// TIA Portal V15.1 export
// export: Created 2024-06-21T08:41:25.4338314Z, ExportSetting WithDefaults, DisplayName Totally Integrated Automation Portal, DisplayVersion V15.1 Update 5, DisplayName TIA Portal Openness, DisplayVersion V15.1 Update 5, DisplayName SINAMICS Startdrive Advanced, DisplayVersion V15.1, DisplayName G130, G150, S120, S150, SINAMICS MV, S210, DisplayVersion V15.1, DisplayName G110M, G120, G120C, G120D, G120P, DisplayVersion V15.1, DisplayName STEP 7 Professional, DisplayVersion V15.1 Update 5, DisplayName STEP 7 Safety, DisplayVersion V15.1, DisplayName WinCC Professional, DisplayVersion V15.1 Update 5, DisplayName SIMATIC Visualization Architect, DisplayVersion V15.1
FUNCTION "209000NCP01ComSafety" : Void   // FC199, FBD
TITLE = 209000NCP01ComSafety
{ S7_Optimized_Access := 'TRUE' }
VERSION : 0.1
// stored: AutoNumber false, IsIECCheckEnabled false, SetENOAutomatically False, UDAEnableTagReadback false
BEGIN

REGION Network 1: **** 5.2 - Equations **** 209230ASD01 Alarm Reset PB
   // Alarm Reset Push Button of MGB
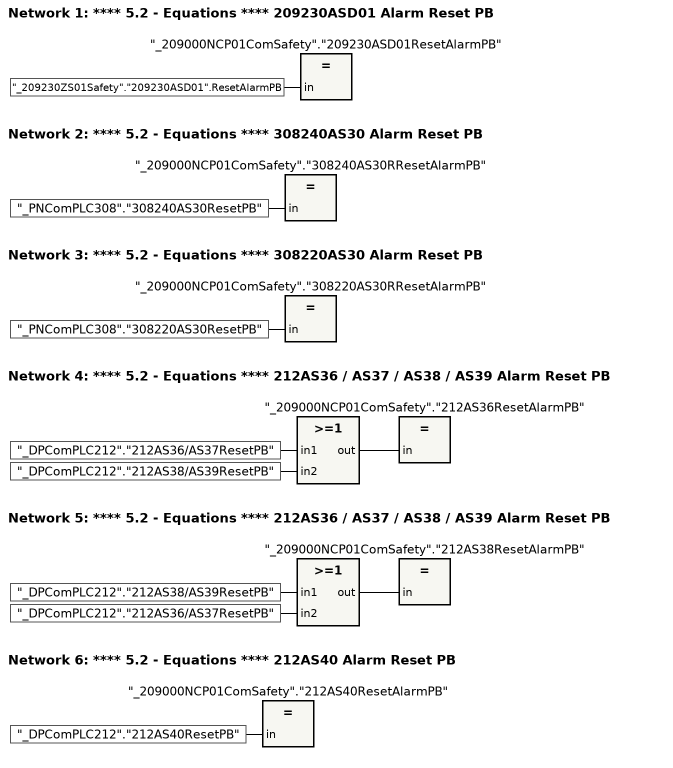
   "_209000NCP01ComSafety"."209230ASD01ResetAlarmPB" := "_209230ZS01Safety"."209230ASD01".ResetAlarmPB;
END_REGION

REGION Network 2: **** 5.2 - Equations **** 308240AS30 Alarm Reset PB
   "_209000NCP01ComSafety"."308240AS30RResetAlarmPB" := "_PNComPLC308"."308240AS30ResetPB";
END_REGION

REGION Network 3: **** 5.2 - Equations **** 308220AS30 Alarm Reset PB
   "_209000NCP01ComSafety"."308220AS30RResetAlarmPB" := "_PNComPLC308"."308220AS30ResetPB";
END_REGION

REGION Network 4: **** 5.2 - Equations **** 212AS36 / AS37 / AS38 / AS39 Alarm Reset PB
   "_209000NCP01ComSafety"."212AS36ResetAlarmPB" := "_DPComPLC212"."212AS36/AS37ResetPB" OR "_DPComPLC212"."212AS38/AS39ResetPB";
END_REGION

REGION Network 5: **** 5.2 - Equations **** 212AS36 / AS37 / AS38 / AS39 Alarm Reset PB
   "_209000NCP01ComSafety"."212AS38ResetAlarmPB" := "_DPComPLC212"."212AS38/AS39ResetPB" OR "_DPComPLC212"."212AS36/AS37ResetPB";
END_REGION

REGION Network 6: **** 5.2 - Equations **** 212AS40 Alarm Reset PB
   "_209000NCP01ComSafety"."212AS40ResetAlarmPB" := "_DPComPLC212"."212AS40ResetPB";
END_REGION
END_FUNCTION
